//Result is TRUE if INT index is out of range
{attribute 'no_check'}
FUNCTION boundsError : BOOL
VAR_INPUT
	Index													:INT;
	Lower													:INT;
	Upper													:INT;
END_VAR                 								
VAR
END_VAR

BoundsError:=index < lower OR index > upper;

END_FUNCTION

(* stored: Version 1.1.0.1, ProductVersion 3.1.4024.3
   POU boundsError: Id {89008b2c-51dd-45be-ab84-2bd03bb522cd}, SpecialFunc None *)
